(* -----------------------------------------------------------------------------
| This sample has been supplied by Beckhoff As-Is and is intended only as an   |
| example implementation. Functionality is not guaranteed.                     |
----------------------------------------------------------------------------- *)

FUNCTION_BLOCK FB_FLM_ReadCmd

VAR_INPUT
	stIn : ST_FLM_In;
	stIotCmd : ST_FLM_Cmd;
END_VAR

VAR_OUTPUT
	stCmd : ST_FLM_Cmd;
END_VAR

VAR_IN_OUT
	
END_VAR

VAR
	fbRtStart	: R_TRIG;
	fbRtStop	: R_TRIG;
	fbTpAck		: TP;	
END_VAR
VAR CONSTANT
	
END_VAR

(* -----------------------------------------------------------------------------
| This sample has been supplied by Beckhoff As-Is and is intended only as an   |
| example implementation. Functionality is not guaranteed.                     |
----------------------------------------------------------------------------- *)

fbRtStart(CLK := stIn.bStartButton OR stIotCmd.bStart);
fbRtStop(CLK := stIn.bStopButton OR stIotCmd.bStop);
fbTpAck(IN:= stIn.bAckButton OR stIotCmd.bAck, PT:= T#200MS);


stCmd.bAck		:= fbTpAck.Q;
stCmd.bStop		:= fbRtStop.Q;
stCmd.bStart	:= fbRtStart.Q;

END_FUNCTION_BLOCK

(* stored: Version 1.1.0.1, ProductVersion 3.1.4024.12
   POU FB_FLM_ReadCmd: Id {3bd6bcbd-b96a-438a-b42e-27669aab7d32}, SpecialFunc None *)
